FUNCTION_BLOCK OutputSender (* Extracted Composite Function Block Type *)
  (* Version 11/3/2016, Dmitry *)
  PACKAGE Main;
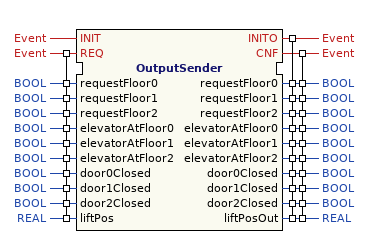
  EVENT_INPUT
    INIT; (* Initialization Request *)
    REQ WITH requestFloor0, requestFloor1, requestFloor2, elevatorAtFloor0, elevatorAtFloor1, elevatorAtFloor2, door0Closed, door1Closed, door2Closed, liftPos; (* Normal Execution Request *)
  END_EVENT
  EVENT_OUTPUT
    INITO WITH requestFloor0, requestFloor1, requestFloor2, elevatorAtFloor0, elevatorAtFloor1, elevatorAtFloor2, door0Closed, door1Closed, door2Closed, liftPosOut; (* Initialization Confirm *)
    CNF WITH requestFloor0, requestFloor1, requestFloor2, elevatorAtFloor0, elevatorAtFloor1, elevatorAtFloor2, door0Closed, door1Closed, door2Closed, liftPosOut; (* Execution Confirmation *)
  END_EVENT
  VAR_INPUT
    requestFloor0 : BOOL;
    requestFloor1 : BOOL;
    requestFloor2 : BOOL;
    elevatorAtFloor0 : BOOL;
    elevatorAtFloor1 : BOOL;
    elevatorAtFloor2 : BOOL;
    door0Closed : BOOL;
    door1Closed : BOOL;
    door2Closed : BOOL;
    liftPos : REAL;
  END_VAR
  VAR_OUTPUT
    requestFloor0 : BOOL;
    requestFloor1 : BOOL;
    requestFloor2 : BOOL;
    elevatorAtFloor0 : BOOL;
    elevatorAtFloor1 : BOOL;
    elevatorAtFloor2 : BOOL;
    door0Closed : BOOL;
    door1Closed : BOOL;
    door2Closed : BOOL;
    liftPosOut : REAL;
  END_VAR
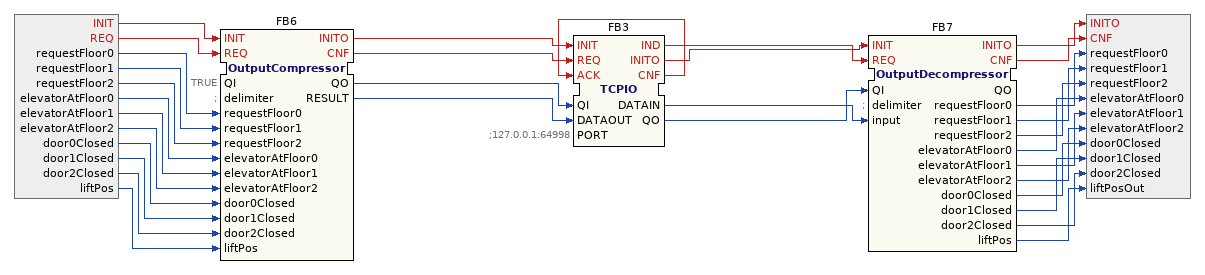
  FBS
    FB3 : TCPIO(PORT := ;127.0.0.1:64998);
    FB7 : OutputDecompressor(delimiter := ;);
    FB6 : OutputCompressor(QI := TRUE, delimiter := ;);
  END_FBS
  EVENT_CONNECTIONS
    FB6.INITO TO FB3.INIT;
    INIT TO FB6.INIT;
    REQ TO FB6.REQ;
    FB6.CNF TO FB3.REQ;
    FB3.IND TO FB7.REQ;
    FB3.INITO TO FB7.INIT;
    FB3.CNF TO FB3.ACK;
    FB7.INITO TO INITO;
    FB7.CNF TO CNF;
  END_CONNECTIONS
  DATA_CONNECTIONS
    FB6.QO TO FB3.QI;
    FB7.requestFloor0 TO requestFloor0;
    FB7.requestFloor1 TO requestFloor1;
    FB7.requestFloor2 TO requestFloor2;
    FB7.elevatorAtFloor0 TO elevatorAtFloor0;
    FB7.elevatorAtFloor1 TO elevatorAtFloor1;
    FB7.elevatorAtFloor2 TO elevatorAtFloor2;
    FB7.door0Closed TO door0Closed;
    FB7.door1Closed TO door1Closed;
    FB7.door2Closed TO door2Closed;
    requestFloor0 TO FB6.requestFloor0;
    requestFloor1 TO FB6.requestFloor1;
    requestFloor2 TO FB6.requestFloor2;
    elevatorAtFloor0 TO FB6.elevatorAtFloor0;
    elevatorAtFloor1 TO FB6.elevatorAtFloor1;
    elevatorAtFloor2 TO FB6.elevatorAtFloor2;
    door0Closed TO FB6.door0Closed;
    door1Closed TO FB6.door1Closed;
    door2Closed TO FB6.door2Closed;
    liftPos TO FB6.liftPos;
    FB3.DATAIN TO FB7.input;
    FB6.RESULT TO FB3.DATAOUT;
    FB3.QO TO FB7.QI;
    FB7.liftPos TO liftPosOut;
  END_CONNECTIONS
END_FUNCTION_BLOCK
